(* MC3 specific settings. Generation independent settings (JogMode) live on
   I_AxisSettings so that generic consumers never touch a Tc3_Mc3Ptp type. *)
INTERFACE I_Mc3Settings EXTENDS I_Base

PROPERTY BufferMode : REFERENCE TO Tc3_Mc3Ptp.EBufferMode
GET
END_GET
END_PROPERTY

PROPERTY Direction : REFERENCE TO Tc3_Mc3Ptp.EModuloDirection
GET
END_GET
END_PROPERTY

END_INTERFACE

(* stored: Version 1.1.0.1, ProductVersion 3.1.4026.20
   Itf I_Mc3Settings: Id {37de20f7-ec83-469c-97f8-33b8f4a87570}
   Property BufferMode: Id {fa76aa55-1427-4930-bb95-00b970d72d34}
   Get Get: Id {1291b058-a331-4617-b351-5b300ed4da32}
   Property Direction: Id {d6610786-db10-424e-87b1-57e8a7f9bbb1}
   Get Get: Id {42ee59a8-0a4a-41e8-afe8-b3a9aecf560c} *)
